TYPE tEncInState1 :
STRUCT
	LatchExternValid		: BIT;
	SetCounterDone			: BIT;
	CounterUnderflow		: BIT;
	CounterOverflow			: BIT;
	ExtrpolationStall		: BIT;
END_STRUCT
END_TYPE

(* stored: Version 1.1.0.1, ProductVersion 3.1.4024.10
   DUT tEncInState1: Id {edbc36c6-d270-4059-ad62-7d95c2adedbe} *)
